(* CoDeSys 2.3 library: 3000SetTickExt.lib *)

(* POU SYSINSTALLTICKHANDLER, ST *)
FUNCTION SYSINSTALLTICKHANDLER : BOOL
VAR_INPUT
	POU:WORD;
	Interval:WORD;
END_VAR
VAR
END_VAR
;
END_FUNCTION
